FUNCTION_BLOCK FB_Carro_DRC_LD
// Transcripción «indirecta» del diagrama de relés y contactos (DRC -> LD)
VAR_INPUT
    ManiobrasTotales: UINT := 2;
    TiempoEspera: TIME := T#2S;
END_VAR
VAR_OUTPUT
    ManiobrasPendientes: UINT;
    TiempoPendiente: TIME;
END_VAR
VAR
    // Estasdos actuales
    EnIzquierda: BOOL;
    
    // Estados futuros
    MarchaDerechaFuturo: BOOL;
    MarchaIzquierdaFuturo: BOOL;
    
    // Bloques funcionales
    FlancoPulsadorMarcha: R_TRIG;
    Intermitencia: FB_Blink;
    TemporizadorEspera: TON;
    ContadorManiobras: CTD := (Q := TRUE);
    
    // Entradas
    i_PulsadorMarcha AT %I*: BOOL;
    i_FinalCarreraIzquierda AT %I*: BOOL := TRUE;
    i_FinalCarreraDerecha AT %I*: BOOL;
    
    // Salidas
    o_MarchaIzquierda AT %I*: BOOL;
    o_MarchaDerecha AT %I*: BOOL;
    o_LamparaMarcha AT %I*: BOOL;
END_VAR

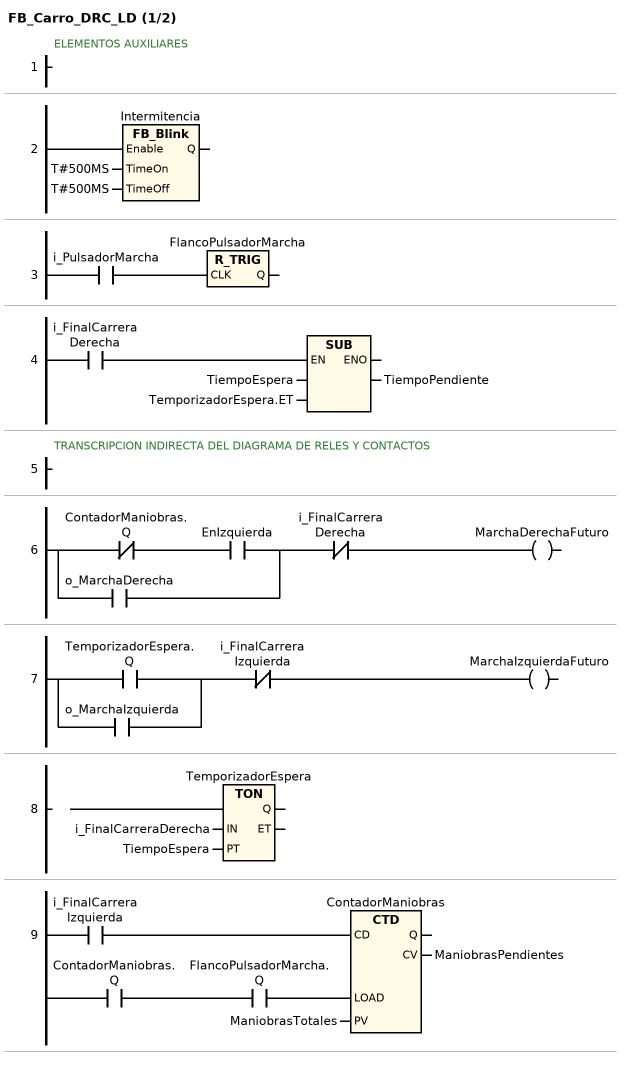
// NETWORK 1
// ELEMENTOS AUXILIARES

// NETWORK 2
Intermitencia(Enable := TRUE, TimeOn := T#500MS, TimeOff := T#500MS); // FB_Blink

// NETWORK 3
FlancoPulsadorMarcha(CLK := i_PulsadorMarcha); // R_TRIG

// NETWORK 4
IF i_FinalCarreraDerecha THEN TiempoPendiente := TiempoEspera - TemporizadorEspera.ET; END_IF

// NETWORK 5
// TRANSCRIPCION INDIRECTA DEL DIAGRAMA DE RELES Y CONTACTOS

// NETWORK 6
MarchaDerechaFuturo := (NOT ContadorManiobras.Q AND EnIzquierda OR o_MarchaDerecha) AND NOT i_FinalCarreraDerecha;

// NETWORK 7
MarchaIzquierdaFuturo := (TemporizadorEspera.Q OR o_MarchaIzquierda) AND NOT i_FinalCarreraIzquierda;

// NETWORK 8
TemporizadorEspera(IN := i_FinalCarreraDerecha, PT := TiempoEspera); // TON

// NETWORK 9
ContadorManiobras(
    CD := i_FinalCarreraIzquierda,
    LOAD := ContadorManiobras.Q AND FlancoPulsadorMarcha.Q,
    PV := ManiobrasTotales,
    CV => ManiobrasPendientes); // CTD

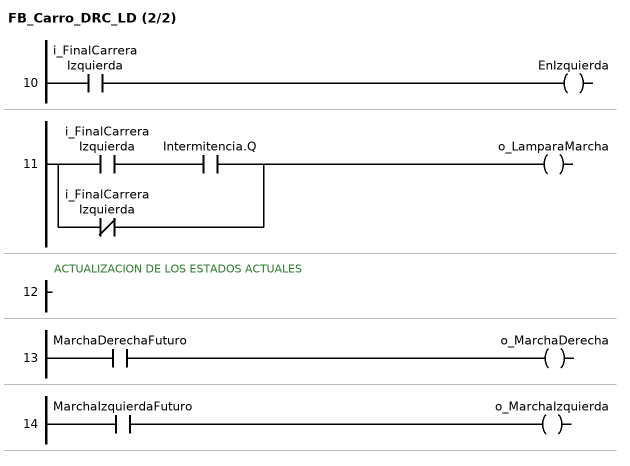
// NETWORK 10
EnIzquierda := i_FinalCarreraIzquierda;

// NETWORK 11
o_LamparaMarcha := i_FinalCarreraIzquierda AND Intermitencia.Q OR NOT i_FinalCarreraIzquierda;

// NETWORK 12
// ACTUALIZACION DE LOS ESTADOS ACTUALES

// NETWORK 13
o_MarchaDerecha := MarchaDerechaFuturo;

// NETWORK 14
o_MarchaIzquierda := MarchaIzquierdaFuturo;

END_FUNCTION_BLOCK

(* stored: Version 1.1.0.1, ProductVersion 3.1.4024.16
   POU FB_Carro_DRC_LD: Id {95007db2-6afe-415c-a00b-f8f7958ae86c}, SpecialFunc None *)
